// TIA Portal V19 export
TYPE "C501_VAR_JPP_TYPIC"
   STRUCT
      BST { ExternalAccessible := 'False'; ExternalVisible := 'False'; ExternalWritable := 'False'} : USInt;   // Bestuurbaarheid
      BSC { ExternalAccessible := 'False'; ExternalVisible := 'False'; ExternalWritable := 'False'} : USInt;   // NOK = Storing aanwezig die beschikbaarheid beinvloed
      PWR { ExternalAccessible := 'False'; ExternalVisible := 'False'; ExternalWritable := 'False'} : Real;   // Actueel vermogen van het pomppaar
      STS { ExternalAccessible := 'False'; ExternalVisible := 'False'; ExternalWritable := 'False'} : USInt;   // Aan = er is minstens een jockeypomp aangeschakeld Uit = alle jockeypompen zijn uit
   END_STRUCT;
END_TYPE
